RoboDK station: Proyecto.rdk

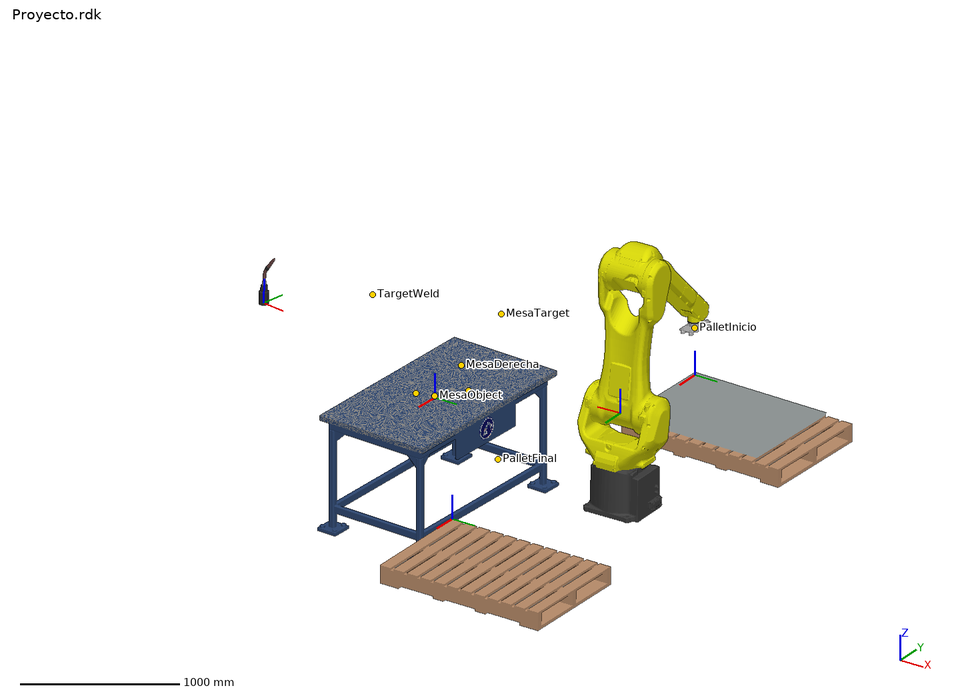
[picture v0: the station drawn from its stored meshes, robots at their saved joint values, targets as dots, program paths as lines]
Station Proyecto (saved by RoboDK 5.3.2). Poses are relative to the parent item; angles as X-Y-Z fixed-axis rotations.
Station parameters (name, value as stored): Pencil, 0, BoolWeld, 0, BoolMove, 1, BoxNumber, 1
  - frame FrameA at (-184.67, 291.95, 650.53) mm, rotated rx -1.31 ry -0.19 rz -8.11 deg
    - target TargetWeld (joint target) at (944.02, -20.21, 373.85) mm, rotated rx 180 ry 0 rz -178.06 deg; joints [-1.968, -11.621, -14.548, -3.444, -40.566, 185.818]
    - object Welding Gun at (0, 0, 0) mm, size 122.1 x 64 x 340.8 mm
  - frame FrameB at (2542.22, 283.32, 650) mm, rotated rx 0 ry 0 rz -178.06 deg
    - robot ROBOTB (model Fanuc M-20iB/25): 6 axes, payload 25 kg, reach 1853 mm, repeatability 0.05 mm, weight 210 kg
        modified DH rows (alpha deg, a mm, theta deg, d mm): 0, 0, 0, 650; -90, 80, -90, 0; 0, 905, 0, 0; -90, 120, 0, 865; 90, 0, 0, 0; -90, 0, 0, 100
        base shift (0, 0, -650) mm
        joint limits [-180, -120, -70, -200, -145, -270] to [180, 120, 230, 200, 145, 270]; home [0, 0, 0, 0, 0, 0]; saved at [-89.529, 5.532, -45.178, 1.834, -45.315, -183.235]
      - tool GripperA, TCP at (0, 0, 30) mm, rotated rx 0 ry 0 rz 90 deg, size 209.9 x 42 x 100 mm, geometry from test.iges
      - tool TCP A, TCP at (0, 0, 37.5) mm, rotated rx 0 ry 0 rz 90 deg
      - tool TCP A, TCP at (0, 0, 37.5) mm, rotated rx 0 ry 0 rz 90 deg
    - frame PalletInicial at (552.9, -1706.9, -579.07) mm, rotated rx 0 ry 0 rz 87.89 deg
      - object Pallet 1200mmx800mm at (0, 0, 0) mm, size 800 x 1200 x 125 mm, geometry from Pallet-1200mmx800mm-Type-1.sld
      - object Square at (0, 0, 0) mm, size 100 x 100 x 0 mm, geometry from Square.sld
      - object Metal_1 at (125, 125, 2.5) mm, size 250 x 250 x 0 mm, geometry from Square.sld
      - object Metal_2 at (375, 125, 2.5) mm, size 250 x 250 x 0 mm, geometry from Square.sld
      - object Metal_3 at (625, 125, 2.5) mm, size 250 x 250 x 0 mm, geometry from Square.sld
      - object Metal_4 at (125, 375, 2.5) mm, size 250 x 250 x 0 mm, geometry from Square.sld
      - object Metal_5 at (375, 375, 2.5) mm, size 250 x 250 x 0 mm, geometry from Square.sld
      - object Metal_6 at (625, 375, 2.5) mm, size 250 x 250 x 0 mm, geometry from Square.sld
      - object Metal_7 at (125, 625, 2.5) mm, size 250 x 250 x 0 mm, geometry from Square.sld
      - object Metal_8 at (375, 625, 2.5) mm, size 250 x 250 x 0 mm, geometry from Square.sld
      - object Metal_9 at (625, 625, 2.5) mm, size 250 x 250 x 0 mm, geometry from Square.sld
      - object Metal_10 at (125, 875, 2.5) mm, size 250 x 250 x 0 mm, geometry from Square.sld
      - object Metal_11 at (375, 875, 2.5) mm, size 250 x 250 x 0 mm, geometry from Square.sld
      - object Metal_12 at (625, 875, 2.5) mm, size 250 x 250 x 0 mm, geometry from Square.sld
      - object Metal_13 at (125, 125, 7.5) mm, size 250 x 250 x 0 mm, geometry from Square.sld
      - object Metal_14 at (375, 125, 7.5) mm, size 250 x 250 x 0 mm, geometry from Square.sld
      - object Metal_15 at (625, 125, 7.5) mm, size 250 x 250 x 0 mm, geometry from Square.sld
      - object Metal_16 at (125, 375, 7.5) mm, size 250 x 250 x 0 mm, geometry from Square.sld
      - object Metal_17 at (375, 375, 7.5) mm, size 250 x 250 x 0 mm, geometry from Square.sld
      - object Metal_18 at (625, 375, 7.5) mm, size 250 x 250 x 0 mm, geometry from Square.sld
      - object Metal_19 at (125, 625, 7.5) mm, size 250 x 250 x 0 mm, geometry from Square.sld
      - object Metal_20 at (375, 625, 7.5) mm, size 250 x 250 x 0 mm, geometry from Square.sld
      - object Metal_21 at (625, 625, 7.5) mm, size 250 x 250 x 0 mm, geometry from Square.sld
      - object Metal_22 at (125, 875, 7.5) mm, size 250 x 250 x 0 mm, geometry from Square.sld
      - object Metal_23 at (375, 875, 7.5) mm, size 250 x 250 x 0 mm, geometry from Square.sld
      - object Metal_24 at (625, 875, 7.5) mm, size 250 x 250 x 0 mm, geometry from Square.sld
      - object Metal_25 at (125, 125, 12.5) mm, size 250 x 250 x 0 mm, geometry from Square.sld
      - object Metal_26 at (375, 125, 12.5) mm, size 250 x 250 x 0 mm, geometry from Square.sld
      - object Metal_27 at (625, 125, 12.5) mm, size 250 x 250 x 0 mm, geometry from Square.sld
      - object Metal_28 at (125, 375, 12.5) mm, size 250 x 250 x 0 mm, geometry from Square.sld
      - object Metal_29 at (375, 375, 12.5) mm, size 250 x 250 x 0 mm, geometry from Square.sld
      - object Metal_30 at (625, 375, 12.5) mm, size 250 x 250 x 0 mm, geometry from Square.sld
      - object Metal_31 at (125, 625, 12.5) mm, size 250 x 250 x 0 mm, geometry from Square.sld
      - object Metal_32 at (375, 625, 12.5) mm, size 250 x 250 x 0 mm, geometry from Square.sld
      - object Metal_33 at (625, 625, 12.5) mm, size 250 x 250 x 0 mm, geometry from Square.sld
      - object Metal_34 at (125, 875, 12.5) mm, size 250 x 250 x 0 mm, geometry from Square.sld
      - object Metal_35 at (375, 875, 12.5) mm, size 250 x 250 x 0 mm, geometry from Square.sld
      - object Metal_36 at (625, 875, 12.5) mm, size 250 x 250 x 0 mm, geometry from Square.sld
      - object Metal_37 at (125, 125, 17.5) mm, size 250 x 250 x 0 mm, geometry from Square.sld
      - object Metal_38 at (375, 125, 17.5) mm, size 250 x 250 x 0 mm, geometry from Square.sld
      - object Metal_39 at (625, 125, 17.5) mm, size 250 x 250 x 0 mm, geometry from Square.sld
      - object Metal_40 at (125, 375, 17.5) mm, size 250 x 250 x 0 mm, geometry from Square.sld
      - object Metal_41 at (375, 375, 17.5) mm, size 250 x 250 x 0 mm, geometry from Square.sld
      - object Metal_42 at (625, 375, 17.5) mm, size 250 x 250 x 0 mm, geometry from Square.sld
      - object Metal_43 at (125, 625, 17.5) mm, size 250 x 250 x 0 mm, geometry from Square.sld
      - object Metal_44 at (375, 625, 17.5) mm, size 250 x 250 x 0 mm, geometry from Square.sld
      - object Metal_45 at (625, 625, 17.5) mm, size 250 x 250 x 0 mm, geometry from Square.sld
      - object Metal_46 at (125, 875, 17.5) mm, size 250 x 250 x 0 mm, geometry from Square.sld
      - object Metal_47 at (375, 875, 17.5) mm, size 250 x 250 x 0 mm, geometry from Square.sld
      - object Metal_48 at (625, 875, 17.5) mm, size 250 x 250 x 0 mm, geometry from Square.sld
      - object Metal_49 at (125, 125, 22.5) mm, size 250 x 250 x 0 mm, geometry from Square.sld
      - object Metal_50 at (375, 125, 22.5) mm, size 250 x 250 x 0 mm, geometry from Square.sld
      - object Metal_51 at (625, 125, 22.5) mm, size 250 x 250 x 0 mm, geometry from Square.sld
      - object Metal_52 at (125, 375, 22.5) mm, size 250 x 250 x 0 mm, geometry from Square.sld
      - object Metal_53 at (375, 375, 22.5) mm, size 250 x 250 x 0 mm, geometry from Square.sld
      - object Metal_54 at (625, 375, 22.5) mm, size 250 x 250 x 0 mm, geometry from Square.sld
      - object Metal_55 at (125, 625, 22.5) mm, size 250 x 250 x 0 mm, geometry from Square.sld
      - object Metal_56 at (375, 625, 22.5) mm, size 250 x 250 x 0 mm, geometry from Square.sld
      - object Metal_57 at (625, 625, 22.5) mm, size 250 x 250 x 0 mm, geometry from Square.sld
      - object Metal_58 at (125, 875, 22.5) mm, size 250 x 250 x 0 mm, geometry from Square.sld
      - object Metal_59 at (375, 875, 22.5) mm, size 250 x 250 x 0 mm, geometry from Square.sld
      - object Metal_60 at (625, 875, 22.5) mm, size 250 x 250 x 0 mm, geometry from Square.sld
    - frame FinalPallet at (716.85, 821.93, -588.16) mm, rotated rx 0 ry 0 rz 88.51 deg
      - object Pallet 1200mmx800mm at (0, 0, 0) mm, size 800 x 1200 x 125 mm, geometry from Pallet-1200mmx800mm-Type-1.sld
    - target PalletInicio (joint target) at (4.06, -861, 239.37) mm, rotated rx -179.57 ry 1.32 rz -1.46 deg; joints [-89.529, 5.532, -45.178, 1.834, -45.315, -183.235] of ROBOTB
    - target MesaDerecha (joint target) at (1330.69, -220.37, -110.68) mm, rotated rx 0 ry 90 rz 85.66 deg; joints [-15.15, 52.494, -57.16, -80.882, -95.84, 57.626] of ROBOTB
    - target MesaTarget (joint target) at (932.33, -67.34, 414.14) mm, rotated rx 180 ry 0 rz 180 deg; joints [-4.131, 3.51, -31.645, 0, -58.355, -85.869] of ROBOTB
    - target MesaObject (joint target) at (1357.74, 37.14, -226.67) mm, rotated rx -179.97 ry -1.31 rz 86.62 deg; joints [1.434, 51.059, -56.792, -2.398, -33.15, 177.197] of ROBOTB
    - target PalletFinal (joint target) at (91.26, 1257.78, 171.79) mm, rotated rx -180 ry 0.01 rz -91.08 deg; joints [85.85, 23.04, -26.67, 0, -63.32, -86.93] of ROBOTB
    - target MesaIzquierda (joint target) at (1348.57, 265.02, -110.81) mm, rotated rx 0 ry -90 rz 85.66 deg; joints [16.484, 54.604, -54.547, 72.79, -101.897, -56.353] of ROBOTB
    - target MesaFrente (joint target) at (1093.79, 59.32, -110.84) mm, rotated rx 90 ry 0 rz 85.66 deg; joints [4.168, 38.837, -76.988, -8.724, 77.133, -178.043] of ROBOTB
  - Python program PrepareSim (listed below)
  - frame Mesa at (1186.39, 200.65, 414.16) mm, rotated rx 0 ry 0 rz -92.4 deg
    - object Table 1400x800x800 at (-417.74, -23.4, 3.44) mm, rotated rx 0 ry 0 rz 0.43 deg, size 1420 x 820 x 800 mm, geometry from Table-1400mmx800mmx800mm.sld
    - object Cube at (0, 0, 0) mm, size 100 x 100 x 100 mm, geometry from box.sld
  - Python program RobotBElementos (listed below)
  - Python program RobotASoldadura (listed below)
  - Python program WeldOn (listed below)
  - Python program BuildBox (listed below)

--- Python program PrepareSim ---
from robolink import *    # RoboDK API
from robodk import *      # Robot toolbox

PARAM_BOOL_WELD= 'BoolWeld'
PARAM_BOOL_MOVE= 'BoolMove'
PARAM_BOX_NUMBER= 'BoxNumber'

RDK = Robolink()

RDK.setParam(PARAM_BOOL_WELD, 0)
RDK.setParam(PARAM_BOOL_MOVE, 0)
RDK.setParam(PARAM_BOX_NUMBER,1)

frame_pallet=RDK.Item('PalletInicial',ITEM_TYPE_FRAME)

def MetalPosition(xs,ys,zs,xp,yp,zp):
    PositionsList=[]
    for k in range(zp):
        for j in range(yp):
            for i in range(xp):
                PositionsList=PositionsList+[[(i+0.5)*xs,(j+0.5)*ys,(k+0.5)*zs]]
    return PositionsList

def MetalSetup(frame,positions,xs,ys,zs):
    n=len(positions)
    for i in range(n):
        newMetal=frame.Paste()
        newMetal.Scale([xs/100,ys/100,zs/100])
        newMetal.setName('Metal_'+str(i+1))
        newMetal.setPose(transl(positions[i]))
        newMetal.setVisible(True, False)
        newMetal.Recolor([0.6719, 0.6953, 0.7031, 1])

def cleanup(objects, startswith="Part "):
    """Deletes all objects where the name starts with "startswith", from the provided list of objects."""
    for item in objects:
        if item.Name().startswith(startswith):
            item.Delete()

#MAIN

RDK.Render(False)
# Elimina los objetos de la simulacion anterior
all_Objects=RDK.ItemList(ITEM_TYPE_OBJECT,False)
cleanup(all_Objects, 'Box_')
cleanup(all_Objects,'Metal_')

all_tools = RDK.ItemList(ITEM_TYPE_TOOL, False)
cleanup(all_tools, 'TCP ')

# Copiar la pieza
Metal=RDK.Item('Square')
Metal.Copy()

# Calculo de posiciones iniciales
positionsXYZ=MetalPosition(250,250,5,3,4,5)
MetalSetup(frame_pallet,positionsXYZ,250,250,5)

RDK.setParam(PARAM_BOOL_MOVE, 1)
RDK.setParam(PARAM_BOOL_WELD, 0)
RDK.RunProgram('WeldOn(RESET)')

RDK.Render(True)

--- Python program RobotBElementos ---
from robolink import *    # RoboDK API
from robodk import *      # Robot toolbox
from time import sleep

RDK = Robolink()

robot =RDK.Item('ROBOTB',ITEM_TYPE_ROBOT)
tool=RDK.Item('GripperA',ITEM_TYPE_TOOL)
frame_pallet=RDK.Item('PalletInicial',ITEM_TYPE_FRAME)
frame_mesa=RDK.Item('Mesa',ITEM_TYPE_FRAME)
frame_pallet_final=RDK.Item('FinalPallet',ITEM_TYPE_FRAME)
target_pallet=RDK.Item('PalletInicio',ITEM_TYPE_TARGET)
target_mesa=RDK.Item('MesaTarget',ITEM_TYPE_TARGET)
target_mesa_Obj=RDK.Item('MesaObject',ITEM_TYPE_TARGET)
target_pallet_final=RDK.Item('PalletFinal',ITEM_TYPE_TARGET)
target_derecha=RDK.Item('MesaDerecha',ITEM_TYPE_TARGET)
target_frente=RDK.Item('MesaFrente',ITEM_TYPE_TARGET)
target_izquierda=RDK.Item('MesaIzquierda',ITEM_TYPE_TARGET)

def MetalPosition(xs,ys,zs,xp,yp,zp):
    PositionsList=[]
    for k in range(zp):
        for j in range(yp):
            for i in range(xp):
                PositionsList=PositionsList+[[(i+0.5)*xs,(j+0.5)*ys,(k+0.5)*zs]]
    return PositionsList

def TCP_On(toolitem):
    """Attaches the closest object to the toolitem Htool pose,
    It will also output appropriate function calls on the generated robot program (call to TCP_On)"""
    toolitem.AttachClosest()
    toolitem.RDK().RunMessage('Set air valve on')
    toolitem.RDK().RunProgram('TCP_On()')

def TCP_Off(toolitem, itemleave=0):
    """Detaches the closest object attached to the toolitem Htool pose,
    It will also output appropriate function calls on the generated robot program (call to TCP_Off)"""
    toolitem.DetachAll(itemleave)
    toolitem.RDK().RunMessage('Set air valve off')
    toolitem.RDK().RunProgram('TCP_Off()')

def BoxPosition(xs,ys,zs,xp,yp,zp):
    PositionsList=[]
    for k in range(zp):
        for j in range(yp):
            for i in range(xp):
                PositionsList=PositionsList+[[(i+0.5)*xs,(j+0.5)*ys,(k)*zs]]
    return PositionsList

#Main
positionsXYZ=MetalPosition(250,250,5,3,4,5)
n = len(positionsXYZ)
i=n-1
BoxPositionXYZ=BoxPosition(250,250,250,3,4,3)

while i>=0:
    tool_xyzrpw = tool.PoseTool()*transl(0,0,7.5)
    tool_tcp = robot.AddTool(tool_xyzrpw, 'TCP A')
    robot.setPoseTool(tool_tcp)
    while RDK.getParam('BoolMove')==0:
        sleep(1)

    # Primera Pieza

    robot.setPoseFrame(frame_pallet)
    MetalPosicion_i = positionsXYZ[i]

    target_i = transl(MetalPosicion_i)*rotx(pi)
    target_i_app = target_i*transl(0,0,2.5)

    robot.MoveJ(target_pallet)

    robot.MoveJ(target_i_app)
    robot.MoveL(target_i)

    TCP_On(tool)
    robot.MoveL(target_i_app)
    robot.MoveJ(target_pallet)

    robot.setPoseFrame(frame_mesa)
    target_pose = transl(0,0,5)*rotx(pi)
    target_app = transl(0,0,7.5)*rotx(pi)

    robot.MoveJ(target_mesa)
    robot.MoveJ(target_app)
    robot.MoveL(target_pose)
    TCP_Off(tool, frame_mesa)
    robot.MoveL(target_app)
    robot.MoveJ(target_mesa)

    i = i - 1

    # Segunda Pieza
    robot.setPoseFrame(frame_pallet)
    MetalPosicion_i = positionsXYZ[i]

    target_i = transl(MetalPosicion_i)*rotx(pi)
    target_i_app = target_i*transl(0,0,2.5)

    robot.MoveJ(target_pallet)

    robot.MoveJ(target_i_app)
    robot.MoveL(target_i)

    TCP_On(tool)
    robot.MoveL(target_i_app)
    robot.MoveJ(target_pallet)

    robot.setPoseFrame(frame_mesa)
    target_pose = transl(-125,0,125)*roty(pi/2)
    target_app = transl(-125,2.5,125)*roty(pi/2)

    robot.MoveJ(target_mesa)
    robot.MoveJ(target_derecha)
    robot.MoveJ(target_app)
    robot.MoveL(target_pose)
    TCP_Off(tool, frame_mesa)
    robot.MoveL(target_app)
    sleep(1)
    RDK.setParam('BoolWeld', 1)
    RDK.setParam('BoolMove', 0)
    while RDK.getParam('BoolMove')==0:
        sleep(1)

    robot.MoveJ(target_derecha)
    robot.MoveJ(target_mesa)

    i = i - 1

    # Tercera Pieza
    robot.setPoseFrame(frame_pallet)
    MetalPosicion_i = positionsXYZ[i]

    target_i = transl(MetalPosicion_i)*rotx(pi)
    target_i_app = target_i*transl(0,0,2.5)

    robot.MoveJ(target_pallet)

    robot.MoveJ(target_i_app)
    robot.MoveL(target_i)

    TCP_On(tool)
    robot.MoveL(target_i_app)
    robot.MoveJ(target_pallet)

    robot.setPoseFrame(frame_mesa)
    target_pose = transl(125,0,125)*roty(-pi/2)
    target_app = transl(125,2.5,125)*roty(-pi/2)

    robot.MoveJ(target_mesa)
    robot.MoveJ(target_izquierda)
    robot.MoveJ(target_app)
    robot.MoveL(target_pose)
    TCP_Off(tool, frame_mesa)
    robot.MoveL(target_app)
    sleep(1)
    RDK.setParam('BoolWeld', 1)
    RDK.setParam('BoolMove', 0)
    while RDK.getParam('BoolMove')==0:
        sleep(1)

    robot.MoveJ(target_izquierda)
    robot.MoveJ(target_mesa)

    i = i - 1

    # Cuarta Pieza
    robot.setPoseFrame(frame_pallet)
    MetalPosicion_i = positionsXYZ[i]

    target_i = transl(MetalPosicion_i)*rotx(pi)
    target_i_app = target_i*transl(0,0,2.5)

    robot.MoveJ(target_pallet)

    robot.MoveJ(target_i_app)
    robot.MoveL(target_i)

    TCP_On(tool)
    robot.MoveL(target_i_app)
    robot.MoveJ(target_pallet)

    robot.setPoseFrame(frame_mesa)
    target_pose = transl(0,125,125)*rotx(pi/2)
    target_app = transl(2.5,125,125)*rotx(pi/2)

    robot.MoveJ(target_mesa)
    robot.MoveJ(target_frente)
    robot.MoveJ(target_app)
    robot.MoveL(target_pose)
    TCP_Off(tool, frame_mesa)
    robot.MoveL(target_app)
    sleep(1)
    RDK.setParam('BoolWeld', 1)
    RDK.setParam('BoolMove', 0)
    while RDK.getParam('BoolMove')==0:
        sleep(1)

    robot.MoveJ(target_frente)
    robot.MoveJ(target_mesa)

    i = i - 1

    # Quinta Pieza
    robot.setPoseFrame(frame_pallet)
    MetalPosicion_i = positionsXYZ[i]

    target_i = transl(MetalPosicion_i)*rotx(pi)
    target_i_app = target_i*transl(0,0,2.5)

    robot.MoveJ(target_pallet)

    robot.MoveJ(target_i_app)
    robot.MoveL(target_i)

    TCP_On(tool)
    robot.MoveL(target_i_app)
    robot.MoveJ(target_pallet)

    robot.setPoseFrame(frame_mesa)
    target_pose = transl(0,0,250)*rotx(pi)
    target_app = transl(0,0,252.5)*rotx(pi)

    robot.MoveJ(target_mesa)
    robot.MoveJ(target_app)
    robot.MoveL(target_pose)
    TCP_Off(tool, frame_mesa)
    robot.MoveL(target_app)
    sleep(1)
    RDK.setParam('BoolWeld', 1)
    RDK.setParam('BoolMove', 0)
    while RDK.getParam('BoolMove')==0:
        sleep(1)
    robot.MoveJ(target_mesa)

    RDK.setParam('BoolWeld', 1)
    RDK.setParam('BoolMove', 0)
    while RDK.getParam('BoolMove')==0:
        sleep(1)

    i = i - 1

    # Construir caja

    RDK.RunProgram('BuildBox')
    RDK.RunProgram('WeldOn(RESET)')
    sleep(1)

    # Caja recogida

    tool_xyzrpw = tool.PoseTool()*transl(0,0,250)
    tool_tcp = robot.AddTool(tool_xyzrpw, 'TCP A')
    robot.setPoseTool(tool_tcp)


    target_pose = transl(0,0,-2.5)*rotx(pi)
    target_app = transl(0,0,0)*rotx(pi)


    robot.MoveJ(target_app)
    robot.MoveL(target_pose)
    TCP_On(tool)
    robot.MoveL(target_app)
    robot.MoveL(target_pose)
    robot.MoveJ(target_mesa)

    # Mover Caja

    robot.MoveJ(target_pallet_final)
    robot.setPoseFrame(frame_pallet_final)
    positionBox=transl(BoxPositionXYZ[int((n-i)/5-1)])*rotx(pi)
    robot.MoveJ(positionBox)

    TCP_Off(tool, frame_pallet_final)

--- Python program RobotASoldadura ---
from robolink import *    # RoboDK API
from robodk import *      # Robot toolbox
from time import sleep

RDK = Robolink()

robot =RDK.Item('ROBOTA',ITEM_TYPE_ROBOT)
frame_mesa=RDK.Item('Mesa',ITEM_TYPE_FRAME)
target_soldar=RDK.Item('TargetWeld',ITEM_TYPE_TARGET)

#Main

#Soldar pieza 1

while True:
    RDK.RunProgram('WeldOn(RESET)')
    sleep(1)
    robot.setSpeed(100,100)
    robot.MoveJ(target_soldar)
    robot.setPoseFrame(frame_mesa)
    while RDK.getParam('BoolWeld')==0:
        sleep(1)

    target_pose_in = transl(-125,-125,5)*roty(-5*pi/6)
    robot.MoveJ(target_pose_in)
    RDK.RunProgram('WeldOn(ON)')
    sleep(1)
    robot.setSpeed(100,100)
    target_pose_fin = transl(-125,125,5)*roty(-5*pi/6)
    robot.MoveL(target_pose_fin)
    RDK.setParam('BoolMove', 1)
    RDK.setParam('BoolWeld', 0)


#Soldar pieza 2
    RDK.RunProgram('WeldOn(OFF)')
    sleep(1)
    robot.setSpeed(100,100)
    robot.MoveJ(target_soldar)
    robot.setPoseFrame(frame_mesa)
    while RDK.getParam('BoolWeld')==0:
        sleep(1)

    target_pose_in = transl(125,125,5)*roty(5.5*pi/6)
    robot.MoveJ(target_pose_in)
    RDK.RunProgram('WeldOn(ON)')
    sleep(1)
    robot.setSpeed(100,100)
    target_pose_fin = transl(125,-125,5)*roty(5.5*pi/6)
    robot.MoveL(target_pose_fin)
    RDK.setParam('BoolMove', 1)
    RDK.setParam('BoolWeld', 0)

    #Soldar pieza 3
    RDK.RunProgram('WeldOn(OFF)')
    sleep(1)
    robot.setSpeed(100,100)
    robot.MoveJ(target_soldar)
    robot.setPoseFrame(frame_mesa)
    while RDK.getParam('BoolWeld')==0:
        sleep(1)

    target_pose_fin = transl(-125,125,250)*rotx(pi/12)*roty(-5*pi/6)
    robot.MoveL(target_pose_fin)
    RDK.RunProgram('WeldOn(ON)')
    sleep(1)
    robot.setSpeed(100,100)
    target_pose_in = transl(-125,125,5)*rotx(pi/12)*roty(-5*pi/6)
    robot.MoveL(target_pose_in)

    target_pose_fin = transl(125,125,5)*rotx(pi/12)*roty(5.5*pi/6)
    robot.MoveL(target_pose_fin)

    target_pose_fin = transl(125,125,250)*rotx(pi/12)*roty(5.5*pi/6)
    robot.MoveL(target_pose_fin)
    RDK.setParam('BoolMove', 1)
    RDK.setParam('BoolWeld', 0)


    #Soldar pieza 4
    RDK.RunProgram('WeldOn(OFF)')
    sleep(1)
    robot.setSpeed(100,100)
    robot.MoveJ(target_soldar)
    robot.setPoseFrame(frame_mesa)
    while RDK.getParam('BoolWeld')==0:
        sleep(1)

    target_pose_in = transl(-125,-125,250)*rotx(pi/12)*roty(5*pi/6)
    robot.MoveJ(target_pose_in)
    RDK.RunProgram('WeldOn(ON)')
    sleep(1)
    robot.setSpeed(100,100)
    target_pose_fin = transl(-125,125,250)*rotx(pi/12)*roty(5*pi/6)
    robot.MoveL(target_pose_fin)

    RDK.RunProgram('WeldOn(OFF)')
    sleep(1)
    robot.setSpeed(100,100)
    robot.MoveJ(target_soldar)
    robot.setPoseFrame(frame_mesa)

    target_pose_fin = transl(125,-125,250)*rotx(pi/12)*roty(-3*pi/6)
    robot.MoveL(target_pose_fin)
    RDK.RunProgram('WeldOn(ON)')
    sleep(1)
    robot.setSpeed(100,100)
    target_pose_fin = transl(125,125,250)*rotx(pi/12)*roty(-3*pi/6)
    robot.MoveL(target_pose_fin)

    RDK.RunProgram('WeldOn(OFF)')
    sleep(1)
    robot.setSpeed(100,100)
    robot.MoveJ(target_soldar)
    robot.setPoseFrame(frame_mesa)
    RDK.setParam('BoolMove', 1)
    RDK.setParam('BoolWeld', 0)

    robot.MoveJ(target_soldar)
    robot.setPoseFrame(frame_mesa)
    while RDK.getParam('BoolWeld')==0:
        sleep(1)


    target_pose_in = transl(-125,125,250)*rotx(7*pi/6)
    robot.MoveJ(target_pose_in)
    RDK.RunProgram('WeldOn(ON)')
    sleep(1)
    robot.setSpeed(100,100)
    target_pose_fin = transl(125,125,250)*rotx(7*pi/6)
    robot.MoveL(target_pose_fin)


    #Retorno
    RDK.RunProgram('WeldOn(OFF)')
    sleep(1)
    robot.setSpeed(100,100)
    robot.MoveJ(target_soldar)
    robot.setPoseFrame(frame_mesa)

    RDK.setParam('BoolMove', 1)
    RDK.setParam('BoolWeld', 0)

--- Python program WeldOn ---
# This macro allows simulating the material deposition of a weld gun
# By default, this macro will activate the trace once it is called.
# Run the macro ArcEnd to stop the trace.
#
# The macros ArcStart, ArcEnd and WeldOn, SpindleOn, all behave in a similar way, the only difference is the default behavior
# This behavior simmulates Fanuc Arc Welding and triggers appropriate output when using the customized post processor.
# Select ESC to clear the trace manually.
#
# It is possible to call WeldOn(ON) to simulate turning the material deposition ON or WeldOn(OFF) to stop simulating the gun
# Calling WeldOn(RESET) clears all displayed data.
# The macro will output spray gun statistics
#
# Optional:
#     This macro can manage multiple guns and multiple colors.
#     As an example, you can call this macro the following way:
#
# WeldOn(State, ToolName, Color)
#     State: [ON/OFF/RESET]
#     TorchName: The name of the tool. For example: Tool 1
#     Color: A named color or a hex color in the format: '#AARRGGBB'
#             Important: for full color definition you should provide Alpha channel first
#
# Examples:
#     WeldOn(ON)                 # Turn on the trace using the default color
#     WeldOn(OFF)                # Turn off the tool trace
#     WeldOn(ON, Tool 1, yellow) # Turn on the trace for tool 1 in yellow
#     WeldOn(ON, Tool 2, blue) # Turn on the trace for tool 2 in blue
#     WeldOn(OFF, Torch1)        # Turn off trace for Torch 1
#     WeldOn(ON, Torch1, #889900FF) # Turn on the trace for torch 2 in a violet color
#     WeldOn(ON, ,red)         # Turn on the trace for a generic torch in red color
#
# --------------------------------------------------------------
# This script shows how to create "spray" object in RoboDK that allows simulating particle deposition by using:
# RDK.Spray_Add(tool, object, options_command, volume, geometry)
#    tool: tool item (TCP) to use
#    object: object to project the particles
#    options_command (optional): string to specify options.
#    volume (optional): Matrix of parameters defining the volume of the spray gun
#    geometry (optional): Matrix of vertices defining the triangles.
#
# More information here:
# https://robodk.com/doc/en/PythonAPI/robolink.html#robolink.Robolink.Spray_Add
# https://robodk.com/doc/en/RoboDK-API.html
#
# The scripts ArcStart, ArcEnd and WeldOn and SpindleOn behave in a similar way, the only difference is the default behavior
# This behavior simmulates Fanuc Arc Welding and triggers appropriate output when using the customized post processor.
# Select ESC to clear the trace manually.
#
# Example scripts that use Spray_Add:
#     SpindleOn / SpindleOff    -> Turn trace On/Off
#     ArcOn / ArcOff            -> Turn trace On/Off
#     SprayOn / SprayOff        -> Simulate a spray given a workspace volume (for painting)
#     WeldOn / WeldOff          -> Support for multiple weld guns
#
#----------------------------------------------------------

# Constant variables for the first parameter:
ACTION_RESET    = -1    # Same as: RESET (clear all traces)
ACTION_OFF      =  0    # Same as: OFF (turn on)
ACTION_ON       =  1    # Same as: ON (turn off)

# Define the default Action (ACTION_OFF to deactivate, ACTION_ON to activate, ACTION_RESET to clear any spray gun/trace)
# Setting it to None will display a message
Action = ACTION_ON

# Define the default color as a named color or as #AARRGGBB (Alpha, Red, Green Blue)
# COLOR = 'blue'
COLOR = '#abb1b3' # AARRGGBB

# Use a specific tool as a spray gun
Tool_Name = "Pencil"    # Use the active tool
#Tool_Name = 'Torch1'

# Use a specific object to project particles:
Object_Name = "Plane"  # Use the first object in the active reference frame
#Object_Name = 'Part'

# --------------------------------------------------
# Program start:
from robolink import *    # API to communicate with RoboDK
from robodk import *      # basic matrix operations
RDK = Robolink()

# quit if we are not in simulation mode
if RDK.RunMode() != RUNMODE_SIMULATE:
    quit()

# Check command input (parameters passed in the call). This is the same as if we were doing a command line call passing parameters.
import sys
if len(sys.argv) > 1:
    Action_str = sys.argv[1].strip().upper()
    if 'ON' in Action_str:
        Action = ACTION_ON
    elif 'OFF' in Action_str:
        Action = ACTION_OFF
    elif 'RESET' in Action_str:
        Action = ACTION_RESET
    else:
        Action = int(Action_str)

    if len(sys.argv) > 2:
        Tool_Name = sys.argv[2].strip()
        if Tool_Name == '':
            Tool_Name = None

        if len(sys.argv) > 3:
            COLOR = sys.argv[3].lower().strip()

# Display summary
print("Applying action: " + str(Action))
print("Using tool: " + str(Tool_Name))
print("Using color: " + COLOR)

# Get any previously added spray gun simulations and display statistics (spray on the part vs spray falling out of the part)
info, data = RDK.Spray_GetStats()
n_sprays = data.size(1)
spray_id = -1
if n_sprays > 0 and Tool_Name is not None:
    spray_id = RDK.getParam(Tool_Name)
    if spray_id is None or Action == ACTION_ON or type(spray_id) == str or spray_id >= n_sprays:
        spray_id = -1

    print("Spray gun statistics:")
    print(info)
    print(data.tr())
    # # Diplay statistics
    # RDK.ShowMessage("Material used: %.1f%%<br>Material waisted: %.1f%%<br>Total particles: %.1f" % (data[1,0],data[2,0],data[3,0]), True)
    # # Clear previous spray
    # RDK.Spray_Clear()


# If the default Action is None, display a message to activate/deactivate the spray gun
if Action is None:
    print('Note: This macro can be called as ArcStart(1) or ArcStart(0) or ArcStart(-1)')
    entry = mbox('Turn gun ON or OFF', ('On', '1'), ('Off', '0'))
    if not entry:
        quit()
    Action = int(entry)

# Apply the desired action
if Action == ACTION_OFF:
    # Turn the gun off
    RDK.Spray_SetState(SPRAY_OFF, spray_id)

elif Action == ACTION_RESET:
    # Clear all spray simulations (same as pressing ESC key)
    RDK.Spray_Clear(spray_id)

elif Action == ACTION_ON:
    # Create a new spray gun object in RoboDK
    # by using RDK.Spray_Add(tool, object, options_command, volume, geometry)
    # tool: tool item (TCP) to use
    # object: object to project the particles
    # options_command (optional): string to specify options. Example:
    #     STEP=AxB: Defines the grid to be projected 1x1 means only one line of particle projection (for example, for welding)
    #     PARTICLE: Defines the shape and size of particle (sphere or particle), unless a specific geometry is provided:
    #       a- SPHERE(radius, facets)
    #       b- SPHERE(radius, facets, scalex, scaley, scalez)
    #       b- CUBE(sizex, sizey, sizez)
    #     RAND=factor: Defines a random factor factor 0 means that the particles are not deposited randomly
    #     ELLYPSE: defines the volume as an ellypse (default)
    #     RECTANGLE: defines the volume as a rectangle
    #     PROJECT: project the particles to the surface (default) (for welding, painting or scanning)
    #     NO_PROJECT: does not project the particles to the surface (for example, for 3D printing)
    #
    # volume (optional): Matrix of parameters defining the volume of the spray gun
    # geometry (optional): Matrix of vertices defining the triangles.

    if spray_id < 0:
        tool = 0    # auto detect active tool
        obj = 0     # auto detect object in active reference frame
        if Tool_Name is not None:
            tool = RDK.Item(Tool_Name, ITEM_TYPE_TOOL)

        if Object_Name is not None:
            obj = RDK.Item(Object_Name, ITEM_TYPE_OBJECT)
        # We can specify a given tool object and/or object
        #robot = RDK.Item("ABB IRB 2600-12/1.85", ITEM_TYPE_ROBOT)
        #tools = robot.Childs()
        #if len(tools) > 0:
        #    tool = tools[0]
        #obj = RDK.Item('object', ITEM_TYPE_OBJECT)

        # Create volume parameters
        options_command = "NO_PROJECT PARTICLE=SPHERE(5,8,1,1,1) STEP=1x0 RAND=0 COLOR=" + COLOR

        spray_id = RDK.Spray_Add(tool, obj, options_command)

    # Remember the ID of the spray gun for later
    if Tool_Name is not None:
        RDK.setParam(Tool_Name, spray_id)

    # Apply the state to activate the trace
    RDK.Spray_SetState(SPRAY_ON, spray_id)

--- Python program BuildBox ---
from robolink import *    # RoboDK API
from robodk import *      # Robot toolbox

RDK = Robolink()
Frame_Mesa=RDK.Item('Mesa',ITEM_TYPE_FRAME)

def cleanup(objects, startswith="Part "):
    """Deletes all objects where the name starts with "startswith", from the provided list of objects."""
    for item in objects:
        if item.Name().startswith(startswith) and item.Parent().Name().startswith('Mesa'):
            item.Delete()


RDK.Render(False)

all_Objects=RDK.ItemList(ITEM_TYPE_OBJECT,False)
cleanup(all_Objects,'Metal_')

# Construir la Caja
Box=RDK.Item('Cube')
Box.Copy()
num=RDK.getParam('BoxNumber')
NewBox=Frame_Mesa.Paste()
NewBox.Scale([250/100,250/100,250/100])
NewBox.setName('Box_'+str(int(num)))
NewBox.setPose(transl([0,0,125]))
NewBox.Recolor([0.6719, 0.6953, 0.7031, 1])
NewBox.setVisible(True, False)

RDK.setParam('BoxNumber',num+1)
RDK.Render(True)
